FUNCTION_BLOCK FB_Component_BasicSlaveAxis_SoE EXTENDS FB_Component_BasicSlaveAxis IMPLEMENTS I_BasicAxis
VAR
    DriveReset  : FB_ResetRoutine_SoEDrive;
    State_Reset : INT;
    HomingInfo  : ST_HomingParams;

END_VAR

METHOD CyclicLogic
DriveReset.Axis := THIS^;
DriveReset.CyclicLogic();

SUPER^.CyclicLogic();
END_METHOD

(*! @summary Clears error flags and error IDs for this component*)
METHOD Reset : BOOL
Reset := FALSE;

IF _Error THEN
    CASE State_Reset OF
        0:
            DriveReset.Execute();
            State_Reset := State_Reset + 10;
            Trace('Drive Reset Called ');

        10:
            IF NOT DriveReset.Busy THEN
                State_Reset := State_Reset + 10;
                Trace('Drive Reset Done ');
            END_IF

        20:
            IF SUPER^.Reset() THEN
                Reset       := TRUE;
                State_Reset := 0;
            END_IF
    END_CASE
ELSE
    IF SUPER^.Reset() THEN
        Reset := TRUE;
    END_IF
END_IF
END_METHOD

END_FUNCTION_BLOCK

(* stored: Version 1.1.0.1
   POU FB_Component_BasicSlaveAxis_SoE: Id {eb4aa2e9-6dd8-433e-9ae3-20bc0f68f3e5}, SpecialFunc None
   Folder I_CyclicFB: Id {09e89170-ea44-4267-817f-a90b7cb16729}
   Folder Methods: Id {b45a449e-e1a2-4333-89e0-dcd1008672e9}
   Folder Properties: Id {dce610d6-07bf-4b1e-8ca7-a968710da596}
   Method CyclicLogic: Id {c0c75779-1e1a-4a4f-945b-bdbe44e159ff}
   Method Reset: Id {c1a961f4-b304-4ef3-a164-2fbb9c515ddd} *)
